{attribute 'qualified_only'}
{attribute 'strict'}
TYPE BagDetectionCmd:
(
	DO_NOTHING := 0,
    GET_RESULT_FROM_CAMERA := 1,
    RESET_CAMERA := 2
);
END_TYPE

(* stored: Version 1.1.0.1, ProductVersion 3.1.4024.12
   DUT BagDetectionCmd: Id {1d27aa8f-820d-463d-8a77-3fb2873b8682} *)
